(* IEC 61131-3 sources: Mizera_Tube/Plc (part 18) *)

LD   GSTMAC.yChSelMask.3
AND  SEL_ASSE.yExtMask.7
OR(
LD   RemContrCMinus
AND  Rem_Combination
)
OR(
LD   RemContrCPlus
AND  Rem_Combination
)
ST   GESTAX33.xSelected

***************************************
* Change REF quota for ABS reference
***************************************
CAL  RTRIG_AX_SEL33(CLK:=GESTAX33.xSelected)
LD   RTRIG_AX_SEL33.Q
JMPCN NoSel33
LD   ActualQtaAbsRef               ** Absolute homing quota
ST   QtaRefAbsSet                  ** Absolute homing quota setting
NoSel33:

LD   GESTAX33.xSelected
AND  %nvel14.0                     * Se Vale 1 ?gestito "Encoder Assoluto" (Da Configura Asse)
AND (
LD   ActualQtaAbsRef               ** Absolute homing quota
NE   QtaRefAbsSet                  ** Absolute homing quota setting
)
JMPCN NoEq33

LD   QtaRefAbsSet                  ** Absolute homing quota setting
ST   ActualQtaAbsRef               ** Absolute homing quota
NoEq33:
***************************************

LD   Pul_Jogp                      ** (gPlc0.4)jog+ pushbutton
OR(
LD   RemContrCPlus
AND  Rem_Combination
)
AND  EnabJogRTCP                   ** Abilita Jog RTCP
ANDN EMER_GEN                      ** M0.10 Emergenza generale
AND  GESTAX33.xSelected
AND  GESTAX33.xCloseLoop
ST   GESTAX33.xJogPlus

LD   Pul_Jogm                      ** (gPlc0.5)jog- pushbutton
OR(
LD   RemContrCMinus
AND  Rem_Combination
)
AND  EnabJogRTCP                   ** Abilita Jog RTCP
ANDN EMER_GEN                      ** M0.10 Emergenza generale
AND  GESTAX33.xSelected
AND  GESTAX33.xCloseLoop
ST   GESTAX33.xJogMinus

LD   %nvel14.0                     * Se Vale 1 ?gestito "Encoder Assoluto" (Da Configura Asse)
ST   GESTAX33.xZeroForced          * Forzamento asse tarato

LD   AxesHeadNoZeroed              ** Assi Testa non riferiti
OR   BlcAvX1_user                  ** M74.0 Blocco avanzamento asse X1 da user.plc
OR   BlcAvY1_user                  ** M74.4 Blocco avanzamento asse Y da user.plc
OR   CMD_HOLDMOVING_CH3.7          ** M202 Hold moving command axis CH3 (bit0=X, bit1=Y...)
OR   (
LD   %PLCmsg8.9
OR   %PLCerr20.21
ANDN GESTAX33.xJogMinus
)
OR   (
LD   %PLCmsg8.10
ANDN GESTAX33.xJogPlus
)
ST   GESTAX33.xHoldMoving          * Richiesta blocco avanzamento

LD   Res_Axes                      ** (gPlc25.1) reset axes disable electric shaft
ST   GESTAX33.xUnlock

LDN  ch3_in_ref                    ** channel 3 in ref
ANDN EnJogRtcp                     ** (gPlc0.18)Abilitazione Jog RTCP tuning
ST   GESTAX33.xEnFIR               * Abilita filtri FIR
ST   GESTAX33.xEnFrComp            ** Abilita friction compensation

LD   ALWAYS_ZERO                   ** PLCFLAGS.0  Flag sempre stato off
ST   GESTAX33.xDisLimiter

LD   %cn0.rc8.3            * ch0 in alarm
OR   %cn3.rc8.3            * ch3 in alarm
OR   EmerINC
ST   GESTAX33.xSetAlarm     ** Forzamento allarme asse

CAL  GESTAX33

LD   JOGrunning                    ** One axis moving in JOG
OR   %ra19.1         * Stato JOG all'interno del canale
ST   JOGrunning                    ** One axis moving in JOG

LD   REFrunning                    ** One axis moving in REF
OR   %ra19.2
ST   REFrunning                    ** One axis moving in REF

LD   INCrunning                    ** One axis moving in INC
OR   %ra19.3
ST   INCrunning                    ** One axis moving in INC

LD   GESTAX33.yDriveNotEn
S    %PLCerr2.8          * Axis 33, drive not enable

LD   %pa9                * Velocit?massima asse
MUL  1000
DIV  60
ST   %ra50               * Limitazione velocita' massima interpolazione

LD   BSG_INC                       ** rg1.2 Selezione modo INC (inc.fissi)
JMPCN SVIX33

LD   %pa59               * Velocit?di Repos
MUL  1000
DIV  60
MUL  AxesOverride                  ** (gPlc16) feed degli assi (%)
DIV  100
ST   %ra50               * Limitazione velocita' massima interpolazione

SVIX33:
NOAX33:

*******************************************************************************
*   C spindle axis (34)
*******************************************************************************
PATH %ax34
PATH %ax_lsref34

***************************************
*   POWER ON (PON)
***************************************
LD   %pa3.31            * Simulato
ORN  %cn3.cc1.8         * Maschera assi associata al canale
OR(
LD   %nvel11            ** 1=Mechatrolink
EQ   1
AND  %ring.drv1.RDD_wStatus.4 * PON
)
OR(
LD   %nvel11            ** 3,4=CANopen, Ecat
EQ   3
)
OR(
LD   %nvel11            ** 3,4=CANopen, Ecat
EQ   4
)
OR  (
LD   I_I_READY_DRIVE_C             ** Ready signal drive C
AND  (
LD   %ax34.nvel11
EQ   0
)
)
ST   Pon_C                         ** PON Axe C

LD  %cn3.cc1.8           * Maschera assi associata al canale 0
JMPCN NOAX34

***
*   LIMIT SWITCH & REFERENCE SWITCH

LD   %lsrefmode
ST   AXLSREF34.x_REF_mode        * 0=use ref switch...

LD   %lsreflevel
ST   AXLSREF34.x_TYPE_LS         * (1=NC, 0=NO)

LD   I_I_FC_C_NEG                  ** C minimumm limit switch
ST   AXLSREF34.x_MIN_LS          * Min Limit switch

LD   I_I_FC_C_POS                  ** C maximun limit switch
ST   AXLSREF34.x_MAX_LS          * Max Limit switch

LD   I_I_INDEX_C                   ** C1 Axis Homing Switch
ST   AXLSREF34.x_REF_S           * Reference switch

CAL  AXLSREF34

LD   AXLSREF34.y_MIN_LS          * Min Limit switch
ST   GESTAX34.xMinusLS           * Negative limit switch

LD   AXLSREF34.y_MAX_LS          * Max Limit switch
ST   GESTAX34.xPlusLS            * Positive limit switch

LD   AXLSREF34.y_REF_S           * Reference switch
ST   GESTAX34.xRefLS             * Reference
***

LD   TON_ABIL.Q          * Abilitazione drives
ANDN TOF_MALARM.Q        * Assi in allarme
AND  Pon                           ** PON
ANDN CMD_C_C1_OPENLOOP.0             ** M204 Open loop (bit0=1 C, bit1=1 C1)
ST   GESTAX34.xCloseLoop

LD   GSTMAC.yChSelMask.3
AND  SEL_ASSE.yExtMask.8
ST   GESTAX34.xSelected

***************************************
* Change REF quota for ABS reference
***************************************
CAL  RTRIG_AX_SEL34(CLK:=GESTAX34.xSelected)
LD   RTRIG_AX_SEL34.Q
JMPCN NoSel34
LD   ActualQtaAbsRef               ** Absolute homing quota
ST   QtaRefAbsSet                  ** Absolute homing quota setting
NoSel34:

LD   GESTAX34.xSelected
AND  %nvel14.0                     * Se Vale 1 ?gestito "Encoder Assoluto" (Da Configura Asse)
AND (
LD   ActualQtaAbsRef               ** Absolute homing quota
NE   QtaRefAbsSet                  ** Absolute homing quota setting
)
JMPCN NoEq34

LD   QtaRefAbsSet                  ** Absolute homing quota setting
ST   ActualQtaAbsRef               ** Absolute homing quota
NoEq34:
***************************************

LD   JOY_C_P					   **(gPlc2.9)Joystik C + selezionato
OR   (
LD   Pul_Jogp                      ** (gPlc0.4)jog+ pushbutton
AND  GESTAX34.xSelected
)
AND  EnabJogRTCP                   ** Abilita Jog RTCP
ANDN EMER_GEN                      ** M0.10 Emergenza generale
ANDN cmd_c_c1_gear_run
AND  GESTAX34.xCloseLoop
ST   GESTAX34.xJogPlus

LD   JOY_C_M                       **(gPlc2.10)Joystik C - selezionato
OR   (
LD   Pul_Jogm                      ** (gPlc0.5)jog- pushbutton
AND  GESTAX34.xSelected
)
AND  EnabJogRTCP                   ** Abilita Jog RTCP
ANDN EMER_GEN                      ** M0.10 Emergenza generale
ANDN cmd_c_c1_gear_run
AND  GESTAX34.xCloseLoop
ST   GESTAX34.xJogMinus

LD   %nvel14.0                     * Se Vale 1 ?gestito "Encoder Assoluto" (Da Configura Asse)
ST   GESTAX34.xZeroForced          * Forzamento asse tarato

LD   GESTAX5.xHoldMoving           * Richiesta blocco avanzamento
OR   BlcAvX1_user                  ** M74.0 Blocco avanzamento asse X1 da user.plc
OR   HoldSafePipeX                 ** (LsPlc26.2) Hold moving for X axis, not allow manual movement in pipe area
OR   AxesHeadNoZeroed              ** Assi Testa non riferiti
OR   CMD_HOLDMOVING_CH3.8          ** M202 Hold moving command axis CH3 (bit0=X, bit1=Y...)
OR   MOVE_AXIS34.yHoldMov
ST   GESTAX34.xHoldMoving          * Richiesta blocco avanzamento

LD   MOVE_AXIS34.yFromPlc
ST   GESTAX34.xFromPlc

LD   Res_Axes                      ** (gPlc25.1) reset axes disable electric shaft
ST   GESTAX34.xUnlock
ST   O_O_RESET_DRIVE_C             ** C axis drive reset (disable electric shaft)

LDN  ch3_in_ref                    ** channel 3 in ref
ANDN EnJogRtcp                     ** (gPlc0.18)Abilitazione Jog RTCP tuning
ST   GESTAX34.xEnFIR               * Abilita filtri FIR
ST   GESTAX34.xEnFrComp            ** Abilita friction compensation

LD   ALWAYS_ONE
ST   GESTAX34.xDisLimiter

LD   %cn0.rc8.3            * ch0 in alarm
OR   %cn3.rc8.3            * ch3 in alarm
OR   EmerINC
ST   GESTAX34.xSetAlarm     ** Forzamento allarme asse

CAL  GESTAX34

LD   GESTAX34.yDriveNotEn
S    %PLCerr2.4                    * Axis 34, drive not enable

LD   %pa9                * Velocit?massima asse
MUL  1000
DIV  60
ST   %ra50               * Limitazione velocita' massima interpolazione

LD   BSG_INC                       ** rg1.2 Selezione modo INC (inc.fissi)
JMPCN SVIX34

LD   %pa59               * Velocit?di Repos
MUL  1000
DIV  60
MUL  AxesOverride                  ** (gPlc16) feed degli assi (%)
DIV  100
ST   %ra50               * Limitazione velocita' massima interpolazione

SVIX34:
NOAX34:
********************************************************************************

**************************
* Acknowledg funzioni "M"
**************************

LD   R_TRIG10000.Q       ** (M0.8)M10000_CN0: Invoca Unit_1 (inizialavorazione)
OR   R_TRIG10001.Q       ** (M0.9)M10001_CN0: Invoca Unit_1 (finelavorazione)
AND  M30000_CN3                    ** M0.5 M30000_CN3: Attendi Servizio per Unit_1[(M10000 iniziolav.) / M10001(finelav.)]
ORN  Z_Z1_SEL                      ** (gPlc13.6)Testa Z + Z1 selezionata
OR(
LDN  PRGRUN_CN0                    ** M0.0 cn0.rc8.0  Programma in corso
ANDN PRGRUN_CN3                    ** M0.2 cn3.rc8.0  Programma in corso
)
R    BlckM30000_CN3                ** Blocco M30000_CN3 con Z_Z1 selezionati

CAL R_TRIG_M30000CN3(CLK=M30000_CN3) ** Fronte Up M30000CN3

LD   R_TRIG_M30000CN3.Q  ** Fronte Up M30000CN3
OR   F_TRIG10000.Q        ** FronteDwn M10000_CN0: Invoca Unit_1 (inizialavorazione)
OR   F_TRIG10001.Q        ** FronteDwn M10001_CN0: Invoca Unit_1 (finelavorazione)
AND  Z_Z1_SEL                      ** (gPlc13.6)Testa Z + Z1 selezionata
S    BlckM30000_CN3                ** Blocco M30000_CN3 con Z_Z1 selezionati

LD   M30000_CN3                    ** M0.5 M30000_CN3: Attendi Servizio per Unit_1[(M10000 iniziolav.) / M10001(finelav.)]
ANDN Z_Z1_SEL                      ** (gPlc13.6)Testa Z + Z1 selezionata
AND(
LDN  M10000_CN0                    ** M0.8 M10000_CN0: Invoca Unit_1 (inizialavorazione)
ANDN M10001_CN0                    ** M0.9 M10001_CN0: Invoca Unit_1 (finelavorazione)
ORN  HEADZSEL                      ** (gPlc13.4)Testa 1 selezionata
)
ANDN CN3_REQ_VYZ_ISO
OR(
LD   M30000_CN3                    ** M0.5 M30000_CN3: Attendi Servizio per Unit_1[(M10000 iniziolav.) / M10001(finelav.)]
AND  Z_Z1_SEL                      ** (gPlc13.6)Testa Z + Z1 selezionata
AND  BlckM30000_CN3                ** Blocco M30000_CN3 con Z_Z1 selezionati
)
OR(
LD   M30010_CN3                    ** M0.6 Sblocco Richiesta servizio (M10000_CN0 inizialavorazione)
AND  Z_Z1_SEL                      ** (gPlc13.6)Testa Z + Z1 selezionata
ANDN M30010_CN3_4                  ** Blocco M30010_CN3_CN4 con Z_Z1 selezionati
)
OR(
LD   M30011_CN3                    ** M0.7 Sblocco Richiesta servizio (M10001_CN0 finelavorazione)
AND  Z_Z1_SEL                      ** (gPlc13.6)Testa Z + Z1 selezionata
ANDN M30011_CN3_4                  ** Blocco M30011_CN3_CN4 con Z_Z1 selezionati
)
OR   GESTCH3.yWaitMFun
OR   Ack_Mfun_UsrM                 ** (gPlc13.13) Unlock M-Functions from User_M
ST   CH3END.xWaitMFun

CAL  CH3END

*******************************************************************************
*******************************************************************************
*   @@@ CH5: GESTIONE CAMBIO PALLET
*******************************************************************************
*******************************************************************************
PATH %cn5

LD   ALWAYS_ONE                    ** PLCFLAGS.1  Flag sempre stato on
ST   GESTCH5.xCmdFromInput

LD   ALWAYS_ONE                    ** PLCFLAGS.1  Flag sempre stato on
ST   GESTCH5.xEscOpCmd

LD   %PLCFLAGS.0
ST   GESTCH5.xSelFromInput        * Disabilita selezioni standard macchina

LD   Op_Mode0.ySelRef
ST   GESTCH5.xSelREF

LD   Op_Mode0.ySelSingRef
ST   GESTCH0.xSingleRef

LD   Op_Mode0.ySelJog
ST   GESTCH5.xSelJOG

LD   Op_Mode0.ySelInc
ST   GESTCH5.xSelINC

LD   Op_Mode0.ySelMdi
* todo
*AND (
*LD   UP_SELCHAN                    ** ui17 Canale selezionato da monitor canale
*EQ   5
*)
ST   GESTCH5.xSelMDI

LD   Op_Mode0.ySelAut
ST   GESTCH5.xSelAUT

LD   Pul_Start                     ** (gPlc0.1)Start pushbutton
ANDN EMER_GEN                      ** M0.10 Emergenza generale
AND (
LD   BCO_PRGRUN                    ** rc8.0  Programma in corso
AND  BCO_PRGINT                    ** rc8.1  Programma interrotto
AND  ch5_in_aut
OR   ch5_in_ref
OR(
 LD   BCI_MDI                       ** rc0.11  Selettore modi operativi su MDI (semiautom)
 AND (
 LD  UP_SELCHAN                                     ** ui17 Canale selezionato da monitor canale
 EQ  5
 )
)
)
ST   GESTCH5.xStart               * comando START al canale (esterno)

LD   Res_Ch0                       ** (gPlc25.3) reset channel 0
ST   GESTCH5.xReset               * comando RESET al canale (esterno)

LD   %PLCFLAGS.0                  ** Condizioni richiesta hold canale 0
OR(
LD   Pul_Stop                      ** (gPlc0.2)Stop pushbutton
AND  BCI_MDI                       ** rc0.11  Selettore modi operativi su MDI (semiautom)
)
ST   GESTCH5.xHold                * comando Hold al canale (esterno)

LD   GESTCH0.xEmer
ST   GESTCH5.xEmer                * comando Emergenza al canale (esterno)

LD   5555
ST   GESTCH5.xPPNumber            * numero part program da eseguire

LD   %PLCFLAGS.0
ST   GESTCH5.xBlkSearch
ST   GESTCH5.xIntBlkSrc           * Forzam. esec. ricerca blocco interna
ST   GESTCH5.xOverstore  * Ab. overstore dopo ricerca blocco (provv.)

LD   ChannelFeedrate               ** feedrate for channel
ST   GESTCH5.xOverride

CAL  GESTCH5

LD   GESTCH5.yProgramRun          * Programma in corso
ST   PRGRUN_CN5                    ** M0.27 cn5.rc8.0  Programma in corso

LD   BCO_STB_GET                   ** rc8.17 Strobe per GET resources
AND  AxStopSincGRP                 ** (gPlc13.11)Assi Fermi per sincronismo GRP[ax]
ST   BCI_ACK_GET                   ** rc0.29  ACK per GET resource

*******************************************************************************
*   Virtual X axis for tube following algorithm
*******************************************************************************
PATH %ax50
PATH %ax_lsref50

LD  %cc1.0           * Maschera assi associata al canale 0
JMPCN NOAX50

LD   ALWAYS_ZERO                        ** PLCFLAGS.0  Flag sempre stato off
ST   GESTAX50.xMinusLS           * Negative limit switch

LD   ALWAYS_ZERO                      ** PLCFLAGS.0  Flag sempre stato off
ST   GESTAX50.xPlusLS            * Positive limit switch

LD   ALWAYS_ZERO                     ** PLCFLAGS.0  Flag sempre stato off
ST   GESTAX50.xRefLS             * Reference
***

LD   TON_ABIL.Q          * Abilitazione drives
ANDN TOF_MALARM.Q        * Assi in allarme
AND  Pon                           ** PON
ST   GESTAX50.xCloseLoop
ST   GESTAX50_xCloseLoop

LD   ALWAYS_ZERO                   ** PLCFLAGS.0  Flag sempre stato off
ST   GESTAX50.xSelected

LD   ALWAYS_ZERO                   ** PLCFLAGS.0  Flag sempre stato off
ST   GESTAX50.xJogPlus

LD   ALWAYS_ZERO                   ** PLCFLAGS.0  Flag sempre stato off
ST   GESTAX50.xJogMinus

LD   CMD_HOLDMOVING_CH5.0          ** M203 Hold moving command axis CH5 (bit0=X, bit1=Y...)
ST   GESTAX50.xHoldMoving          * Richiesta blocco avanzamento

LD   ALWAYS_ONE                    ** PLCFLAGS.1  Flag sempre stato on
ST   GESTAX50.xZeroForced          * Forzamento asse tarato
ST   GESTAX50.xLockRef    * Blocco avvio ciclo REF da canale

LD   Res_Axes                      ** (gPlc25.1) reset axes disable electric shaft
ST   GESTAX50.xUnlock

LDN  ch5_in_ref                    ** channel 5 in ref
ANDN EnJogRtcp                     ** (gPlc0.18)Abilitazione Jog RTCP tuning
ST   GESTAX50.xEnFIR               * Abilita filtri FIR
ST   GESTAX50.xEnFrComp            ** Abilita friction compensation

LD   ALWAYS_ONE                   ** PLCFLAGS.0  Flag sempre stato off
ST   GESTAX50.xDisLimiter

LD   %cn0.rc8.3            * ch0 in alarm
OR   %cn3.rc8.3            * ch3 in alarm
OR   EmerINC
ST   GESTAX50.xSetAlarm     ** Forzamento allarme asse

CAL  GESTAX50

LD   JOGrunning                    ** One axis moving in JOG
OR   %ra19.1         * Stato JOG all'interno del canale
ST   JOGrunning                    ** One axis moving in JOG

LD   REFrunning                    ** One axis moving in REF
OR   %ra19.2
ST   REFrunning                    ** One axis moving in REF

LD   INCrunning                    ** One axis moving in INC
OR   %ra19.3
ST   INCrunning                    ** One axis moving in INC

LD   %pa9                * Velocit?massima asse
MUL  1000
DIV  60
ST   %ra50               * Limitazione velocita' massima interpolazione

LD   BSG_INC                       ** rg1.2 Selezione modo INC (inc.fissi)
JMPCN SVIX50

LD   %pa59               * Velocit?di Repos
MUL  1000
DIV  60
MUL  AxesOverride                  ** (gPlc16) feed degli assi (%)
DIV  100
ST   %ra50               * Limitazione velocita' massima interpolazione

SVIX50:
NOAX50:

*******************************************************************************
*   Support 1 follower
*******************************************************************************
PATH %ax51
PATH %ax_lsref51

***************************************
*   POWER ON (PON)
***************************************
LD   %pa3.31            * Simulato
ORN  %cc1.1             * Maschera assi associata al canale
OR(
LD   %nvel11            ** 1=Mechatrolink
EQ   1
AND  %ring.drv1.RDD_wStatus.4 * PON
)
OR(
LD   %nvel11            ** 3,4=CANopen, Ecat
EQ   3
)
OR(
LD   %nvel11            ** 3,4=CANopen, Ecat
EQ   4
)
ST   Pon_Z_Follow            ** PON Axe X_T1

LD  %cc1.1           * Maschera assi associata al canale 0
JMPCN NOAX51

***
*   LIMIT SWITCH & REFERENCE SWITCH

LD   %lsrefmode
ST   AXLSREF51.x_REF_mode        * 0=use ref switch...

LD   %lsreflevel
ST   AXLSREF51.x_TYPE_LS         * (1=NC, 0=NO)

LD   I_I_FC_Z1_SUP_NEG
ST   AXLSREF51.x_MIN_LS          * Min Limit switch

LD   I_I_FC_Z1_SUP_POS           * C saw minimumm limit switch
ST   AXLSREF51.x_MAX_LS          * Max Limit switch

LD   ALWAYS_ZERO                   ** PLCFLAGS.0  Flag sempre stato off
ST   AXLSREF51.x_REF_S           * Reference switch

CAL  AXLSREF51

LD   AXLSREF51.y_MIN_LS          * Min Limit switch
ST   GESTAX51.xMinusLS           * Negative limit switch

LD   AXLSREF51.y_MAX_LS          * Max Limit switch
ST   GESTAX51.xPlusLS            * Positive limit switch

LD   AXLSREF51.y_REF_S           * Reference switch
ST   GESTAX51.xRefLS             * Reference
***

LD   TON_ABIL.Q          * Abilitazione drives
ANDN TOF_MALARM.Q        * Assi in allarme
AND  Pon                           ** PON
ST   GESTAX51.xCloseLoop

LD   GSTMAC.yChSelMask.5
AND  SEL_ASSE.yExtMask.1
ST   GESTAX51.xSelected

***************************************
* Change REF quota for ABS reference
***************************************
CAL  RTRIG_AX_SEL51(CLK:=GESTAX51.xSelected)
LD   RTRIG_AX_SEL51.Q
JMPCN NoSel51
LD   ActualQtaAbsRef               ** Absolute homing quota
ST   QtaRefAbsSet                  ** Absolute homing quota setting
NoSel51:

LD   GESTAX51.xSelected
AND  %nvel14.0                     * Se Vale 1 ?gestito "Encoder Assoluto" (Da Configura Asse)
AND (
LD   ActualQtaAbsRef               ** Absolute homing quota
NE   QtaRefAbsSet                  ** Absolute homing quota setting
)
JMPCN NoEq51

LD   QtaRefAbsSet                  ** Absolute homing quota setting
ST   ActualQtaAbsRef               ** Absolute homing quota
NoEq51:

LD   Pul_Jogp                      ** (gPlc0.4)jog+ pushbutton
AND  GESTAX51.xSelected
AND  EnabJogRTCP                   ** Abilita Jog RTCP
ANDN EMER_GEN                      ** M0.10 Emergenza generale
AND  GESTAX51.xCloseLoop
ST   GESTAX51.xJogPlus

LD   Pul_Jogm                      ** (gPlc0.5)jog- pushbutton
AND  GESTAX51.xSelected
AND  EnabJogRTCP                   ** Abilita Jog RTCP
ANDN EMER_GEN                      ** M0.10 Emergenza generale
AND  GESTAX51.xCloseLoop
ST   GESTAX51.xJogMinus

LDN  %ra3.2
OR   %ra0.9
AND  %ra3.13
ST   Supp_51_GoUp

LD   CMD_HOLDMOVING_CH5.1            ** M203 Hold moving command axis CH5 (bit0=X, bit1=Y...)
ST   GESTAX51.xHoldMoving          * Richiesta blocco avanzamento

LD   %nvel14.0                     * Se Vale 1 ?gestito "Encoder Assoluto" (Da Configura Asse)
ST   GESTAX51.xZeroForced          * Forzamento asse tarato

LD   Res_Axes                      ** (gPlc25.1) reset axes disable electric shaft
ST   GESTAX51.xUnlock

LDN  ch5_in_ref                    ** channel 5 in ref
ANDN EnJogRtcp                     ** (gPlc0.18)Abilitazione Jog RTCP tuning
ST   GESTAX51.xEnFIR               * Abilita filtri FIR
ST   GESTAX51.xEnFrComp            ** Abilita friction compensation

LD   ALWAYS_ONE
ST   GESTAX51.xDisLimiter

LD   %cn0.rc8.3                    * ch0 in alarm
OR   %cn3.rc8.3                    * ch3 in alarm
OR   EmerINC
ST   GESTAX51.xSetAlarm            ** Forzamento allarme asse

LD   GRANT5.1
ST   GESTAX51.xFromPlc

CAL  GESTAX51

LD   JOGrunning                    ** One axis moving in JOG
OR   %ra19.1                       * Stato JOG all'interno del canale
ST   JOGrunning                    ** One axis moving in JOG

LD   REFrunning                    ** One axis moving in REF
OR   %ra19.2
ST   REFrunning                    ** One axis moving in REF

LD   INCrunning                    ** One axis moving in INC
OR   %ra19.3
ST   INCrunning                    ** One axis moving in INC

LD   GESTAX51.yDriveNotEn
S    %PLCerr2.15                   * Axis 52, drive not enable

LD   %pa9                          * Velocit?massima asse
MUL  1000
DIV  60
ST   %ra50                         * Limitazione velocita' massima interpolazione

LD   BSG_INC                       ** rg1.2 Selezione modo INC (inc.fissi)
JMPCN SVIX51

LD   %pa59                         * Velocit?di Repos
MUL  1000
DIV  60
MUL  AxesOverride                  ** (gPlc16) feed degli assi (%)
DIV  100
ST   %ra50                         * Limitazione velocita' massima interpolazione

SVIX51:
NOAX51:

* Z 1 real axis for the pipe following algorithm

PATH %ax52
PATH %ax_lsref52

***************************************
*   POWER ON (PON)
***************************************
LD   %pa3.31            * Simulato
ORN  %cc1.2             * Maschera assi associata al canale
OR(
LD   %nvel11            ** 1=Mechatrolink
EQ   1
AND  %ring.drv1.RDD_wStatus.4 * PON
)
OR(
LD   %nvel11            ** 3,4=CANopen, Ecat
EQ   3
)
OR(
LD   %nvel11            ** 3,4=CANopen, Ecat
EQ   4
)
ST   Pon_Z_Follow2            ** PON Axe X_T1

LD  %cc1.2           * Maschera assi associata al canale 0
JMPCN NOAX52

***
*   LIMIT SWITCH & REFERENCE SWITCH

LD   %lsrefmode
ST   AXLSREF52.x_REF_mode        * 0=use ref switch...

LD   %lsreflevel
ST   AXLSREF52.x_TYPE_LS         * (1=NC, 0=NO)

LD   I_I_FC_Z2_SUP_NEG
ST   AXLSREF52.x_MIN_LS          * Min Limit switch

LD   I_I_FC_Z2_SUP_POS           * C saw maximun limit switch
ST   AXLSREF52.x_MAX_LS          * Max Limit switch

LD   ALWAYS_ZERO                   ** PLCFLAGS.0  Flag sempre stato off
ST   AXLSREF52.x_REF_S           * Reference switch

CAL  AXLSREF52

LD   AXLSREF52.y_MIN_LS          * Min Limit switch
ST   GESTAX52.xMinusLS           * Negative limit switch

LD   AXLSREF52.y_MAX_LS          * Max Limit switch
ST   GESTAX52.xPlusLS            * Positive limit switch

LD   AXLSREF52.y_REF_S           * Reference switch
ST   GESTAX52.xRefLS             * Reference
***

LD   TON_ABIL.Q          * Abilitazione drives
ANDN TOF_MALARM.Q        * Assi in allarme
AND  Pon                           ** PON
ST   GESTAX52.xCloseLoop

LD   GSTMAC.yChSelMask.5
AND  SEL_ASSE.yExtMask.2
ST   GESTAX52.xSelected

***************************************
* Change REF quota for ABS reference
***************************************
CAL  RTRIG_AX_SEL52(CLK:=GESTAX52.xSelected)
LD   RTRIG_AX_SEL52.Q
JMPCN NoSel52
LD   ActualQtaAbsRef               ** Absolute homing quota
ST   QtaRefAbsSet                  ** Absolute homing quota setting
NoSel52:

LD   GESTAX52.xSelected
AND  %nvel14.0                     * Se Vale 1 ?gestito "Encoder Assoluto" (Da Configura Asse)
AND (
LD   ActualQtaAbsRef               ** Absolute homing quota
NE   QtaRefAbsSet                  ** Absolute homing quota setting
)
JMPCN NoEq52

LD   QtaRefAbsSet                  ** Absolute homing quota setting
ST   ActualQtaAbsRef               ** Absolute homing quota
NoEq52:
***************************************

LD   Pul_Jogp                      ** (gPlc0.4)jog+ pushbutton
AND  GESTAX52.xSelected
AND  EnabJogRTCP                   ** Abilita Jog RTCP
ANDN EMER_GEN                      ** M0.10 Emergenza generale
AND  GESTAX52.xCloseLoop
ST   GESTAX52.xJogPlus

LD   Pul_Jogm                      ** (gPlc0.5)jog- pushbutton
AND  GESTAX52.xSelected
AND  EnabJogRTCP                   ** Abilita Jog RTCP
ANDN EMER_GEN                      ** M0.10 Emergenza generale
AND  GESTAX52.xCloseLoop
ST   GESTAX52.xJogMinus

LDN  %ra3.2
OR   %ra0.9
AND  %ra3.13
ST   Supp_52_GoUp

LD   CMD_HOLDMOVING_CH5.2            ** M203 Hold moving command axis CH5 (bit0=X, bit1=Y...)
ST   GESTAX52.xHoldMoving          * Richiesta blocco avanzamento

LD   %nvel14.0                     * Se Vale 1 ?gestito "Encoder Assoluto" (Da Configura Asse)
ST   GESTAX52.xZeroForced          * Forzamento asse tarato

LD   Res_Axes                      ** (gPlc25.1) reset axes disable electric shaft
ST   GESTAX52.xUnlock

LDN  ch5_in_ref                    ** channel 5 in ref
ANDN EnJogRtcp                     ** (gPlc0.18)Abilitazione Jog RTCP tuning
ST   GESTAX52.xEnFIR               * Abilita filtri FIR
ST   GESTAX52.xEnFrComp            ** Abilita friction compensation

LD   ALWAYS_ONE
ST   GESTAX52.xDisLimiter

LD   %cn0.rc8.3            * ch0 in alarm
OR   %cn3.rc8.3            * ch3 in alarm
OR   EmerINC
ST   GESTAX52.xSetAlarm     ** Forzamento allarme asse

LD   GRANT5.2
ST   GESTAX52.xFromPlc

CAL  GESTAX52

LD   JOGrunning                    ** One axis moving in JOG
OR   %ra19.1         * Stato JOG all'interno del canale
ST   JOGrunning                    ** One axis moving in JOG

LD   REFrunning                    ** One axis moving in REF
OR   %ra19.2
ST   REFrunning                    ** One axis moving in REF

LD   INCrunning                    ** One axis moving in INC
OR   %ra19.3
ST   INCrunning                    ** One axis moving in INC

LD   GESTAX52.yDriveNotEn
S    %PLCerr2.14                    * Axis 52, drive not enable

LD   %pa9                * Velocit?massima asse
MUL  1000
DIV  60
ST   %ra50               * Limitazione velocita' massima interpolazione

LD   BSG_INC                       ** rg1.2 Selezione modo INC (inc.fissi)
JMPCN SVIX52

LD   %pa59               * Velocit?di Repos
MUL  1000
DIV  60
MUL  AxesOverride                  ** (gPlc16) feed degli assi (%)
DIV  100
ST   %ra50               * Limitazione velocita' massima interpolazione

SVIX52:
NOAX52:

* Z 3 real axis for the pipe following algorithm

PATH %ax53
PATH %ax_lsref53

***************************************
*   POWER ON (PON)
***************************************
LD   %pa3.31            * Simulato
ORN  %cc1.2             * Maschera assi associata al canale
OR(
LD   %nvel11            ** 1=Mechatrolink
EQ   1
AND  %ring.drv1.RDD_wStatus.4 * PON
)
OR(
LD   %nvel11            ** 3,4=CANopen, Ecat
EQ   3
)
OR(
LD   %nvel11            ** 3,4=CANopen, Ecat
EQ   4
)
OR  (
LD   I_I_READY_DRIVE_Z_FOLL        ** Ready signal drive Z_follower
AND  (
LD   %ax52.nvel11
EQ   0
)
)
ST   Pon_Z_Follow3           ** PON Axe X_T1

LD  %cc1.3           * Maschera assi associata al canale 0
JMPCN NOAX53

***
*   LIMIT SWITCH & REFERENCE SWITCH

LD   %lsrefmode
ST   AXLSREF53.x_REF_mode        * 0=use ref switch...

LD   %lsreflevel
ST   AXLSREF53.x_TYPE_LS         * (1=NC, 0=NO)

LD   I_I_FC_Z3_SUP_NEG                   ** PLCFLAGS.0  Flag sempre stato off
ST   AXLSREF53.x_MIN_LS          * Min Limit switch

LD   I_I_FC_Z3_SUP_POS           * C saw maximun limit switch
ST   AXLSREF53.x_MAX_LS          * Max Limit switch

LD   ALWAYS_ZERO                   ** PLCFLAGS.0  Flag sempre stato off
ST   AXLSREF53.x_REF_S           * Reference switch

CAL  AXLSREF53

LD   AXLSREF53.y_MIN_LS          * Min Limit switch
ST   GESTAX53.xMinusLS           * Negative limit switch

LD   AXLSREF53.y_MAX_LS          * Max Limit switch
ST   GESTAX53.xPlusLS            * Positive limit switch

LD   AXLSREF53.y_REF_S           * Reference switch
ST   GESTAX53.xRefLS             * Reference
***

LD   TON_ABIL.Q          * Abilitazione drives
ANDN TOF_MALARM.Q        * Assi in allarme
AND  Pon                           ** PON
ST   GESTAX53.xCloseLoop

LD   GSTMAC.yChSelMask.5
AND  SEL_ASSE.yExtMask.3
ST   GESTAX53.xSelected

***************************************
* Change REF quota for ABS reference
***************************************
CAL  RTRIG_AX_SEL53(CLK:=GESTAX53.xSelected)
LD   RTRIG_AX_SEL53.Q
JMPCN NoSel53
LD   ActualQtaAbsRef               ** Absolute homing quota
ST   QtaRefAbsSet                  ** Absolute homing quota setting
NoSel53:

LD   GESTAX53.xSelected
AND  %nvel14.0                     * Se Vale 1 ?gestito "Encoder Assoluto" (Da Configura Asse)
AND (
LD   ActualQtaAbsRef               ** Absolute homing quota
NE   QtaRefAbsSet                  ** Absolute homing quota setting
)
JMPCN NoEq53

LD   QtaRefAbsSet                  ** Absolute homing quota setting
ST   ActualQtaAbsRef               ** Absolute homing quota
NoEq53:
***************************************

LD   Pul_Jogp                      ** (gPlc0.4)jog+ pushbutton
AND  GESTAX53.xSelected
AND  EnabJogRTCP                   ** Abilita Jog RTCP
ANDN EMER_GEN                      ** M0.10 Emergenza generale
AND  GESTAX53.xCloseLoop
ST   GESTAX53.xJogPlus

LD   Pul_Jogm                      ** (gPlc0.5)jog- pushbutton
AND  GESTAX53.xSelected
AND  EnabJogRTCP                   ** Abilita Jog RTCP
ANDN EMER_GEN                      ** M0.10 Emergenza generale
AND  GESTAX53.xCloseLoop
ST   GESTAX53.xJogMinus

LDN  %ra3.2
OR   %ra0.9
AND  %ra3.13
ST   Supp_53_GoUp

LD   CMD_HOLDMOVING_CH5.3            ** M203 Hold moving command axis CH5 (bit0=X, bit1=Y...)
ST   GESTAX53.xHoldMoving          * Richiesta blocco avanzamento

LD   %nvel14.0                     * Se Vale 1 ?gestito "Encoder Assoluto" (Da Configura Asse)
ST   GESTAX53.xZeroForced          * Forzamento asse tarato

LD   Res_Axes                      ** (gPlc25.1) reset axes disable electric shaft
ST   GESTAX53.xUnlock

LDN  ch5_in_ref                    ** channel 5 in ref
ANDN EnJogRtcp                     ** (gPlc0.18)Abilitazione Jog RTCP tuning
ST   GESTAX53.xEnFIR               * Abilita filtri FIR
ST   GESTAX53.xEnFrComp            ** Abilita friction compensation

LD   ALWAYS_ONE
ST   GESTAX53.xDisLimiter

LD   %cn0.rc8.3            * ch0 in alarm
OR   %cn3.rc8.3            * ch3 in alarm
OR   EmerINC
ST   GESTAX53.xSetAlarm     ** Forzamento allarme asse

LD   GRANT5.3
ST   GESTAX53.xFromPlc

CAL  GESTAX53

LD   JOGrunning                    ** One axis moving in JOG
OR   %ra19.1         * Stato JOG all'interno del canale
ST   JOGrunning                    ** One axis moving in JOG

LD   REFrunning                    ** One axis moving in REF
OR   %ra19.2
ST   REFrunning                    ** One axis moving in REF

LD   INCrunning                    ** One axis moving in INC
OR   %ra19.3
ST   INCrunning                    ** One axis moving in INC

LD   GESTAX53.yDriveNotEn
S    %PLCerr2.17                   * Axis 53, drive not enable

LD   %pa9                * Velocit?massima asse
MUL  1000
DIV  60
ST   %ra50               * Limitazione velocita' massima interpolazione

LD   BSG_INC                       ** rg1.2 Selezione modo INC (inc.fissi)
JMPCN SVIX53

LD   %pa59               * Velocit?di Repos
MUL  1000
DIV  60
MUL  AxesOverride                  ** (gPlc16) feed degli assi (%)
DIV  100
ST   %ra50               * Limitazione velocita' massima interpolazione

SVIX53:
NOAX53:

* Z 4 real axis for the pipe following algorithm

PATH %ax54
PATH %ax_lsref54

***************************************
*   POWER ON (PON)
***************************************
LD   %pa3.31            * Simulato
ORN  %cc1.4             * Maschera assi associata al canale
OR(
LD   %nvel11            ** 1=Mechatrolink
EQ   1
AND  %ring.drv1.RDD_wStatus.4 * PON
)
OR(
LD   %nvel11            ** 3,4=CANopen, Ecat
EQ   3
)
OR(
LD   %nvel11            ** 3,4=CANopen, Ecat
EQ   4
)
ST   Pon_Z_Follow4           ** PON Axe X_T1

LD  %cc1.4           * Maschera assi associata al canale 0
JMPCN NOAX54

***
*   LIMIT SWITCH & REFERENCE SWITCH

LD   %lsrefmode
ST   AXLSREF54.x_REF_mode        * 0=use ref switch...

LD   %lsreflevel
ST   AXLSREF54.x_TYPE_LS         * (1=NC, 0=NO)

LD   I_I_FC_Z4_SUP_NEG                   ** PLCFLAGS.0  Flag sempre stato off
ST   AXLSREF54.x_MIN_LS          * Min Limit switch

LD   I_I_FC_Z4_SUP_POS           * C saw minimumm limit switch
ST   AXLSREF54.x_MAX_LS          * Max Limit switch

LD   ALWAYS_ZERO                   ** PLCFLAGS.0  Flag sempre stato off
ST   AXLSREF54.x_REF_S           * Reference switch

CAL  AXLSREF54

LD   AXLSREF54.y_MIN_LS          * Min Limit switch
ST   GESTAX54.xMinusLS           * Negative limit switch

LD   AXLSREF54.y_MAX_LS          * Max Limit switch
ST   GESTAX54.xPlusLS            * Positive limit switch

LD   AXLSREF54.y_REF_S           * Reference switch
ST   GESTAX54.xRefLS             * Reference
***

LD   TON_ABIL.Q          * Abilitazione drives
ANDN TOF_MALARM.Q        * Assi in allarme
AND  Pon                           ** PON
ST   GESTAX54.xCloseLoop

LD   GSTMAC.yChSelMask.5
AND  SEL_ASSE.yExtMask.4
ST   GESTAX54.xSelected

***************************************
* Change REF quota for ABS reference
***************************************
CAL  RTRIG_AX_SEL54(CLK:=GESTAX54.xSelected)
LD   RTRIG_AX_SEL54.Q
JMPCN NoSel54
LD   ActualQtaAbsRef               ** Absolute homing quota
ST   QtaRefAbsSet                  ** Absolute homing quota setting
NoSel54:

LD   GESTAX54.xSelected
AND  %nvel14.0                     * Se Vale 1 ?gestito "Encoder Assoluto" (Da Configura Asse)
AND (
LD   ActualQtaAbsRef               ** Absolute homing quota
NE   QtaRefAbsSet                  ** Absolute homing quota setting
)
JMPCN NoEq54

LD   QtaRefAbsSet                  ** Absolute homing quota setting
ST   ActualQtaAbsRef               ** Absolute homing quota
NoEq54:
***************************************

LD   Pul_Jogp                      ** (gPlc0.4)jog+ pushbutton
AND  GESTAX54.xSelected
AND  EnabJogRTCP                   ** Abilita Jog RTCP
ANDN EMER_GEN                      ** M0.10 Emergenza generale
AND  GESTAX54.xCloseLoop
ST   GESTAX54.xJogPlus

LD   Pul_Jogm                      ** (gPlc0.5)jog- pushbutton
AND  GESTAX54.xSelected
AND  EnabJogRTCP                   ** Abilita Jog RTCP
ANDN EMER_GEN                      ** M0.10 Emergenza generale
AND  GESTAX54.xCloseLoop
ST   GESTAX54.xJogMinus

LD   CMD_HOLDMOVING_CH5.4            ** M203 Hold moving command axis CH5 (bit0=X, bit1=Y...)
ST   GESTAX54.xHoldMoving          * Richiesta blocco avanzamento

LD   %nvel14.0                     * Se Vale 1 ?gestito "Encoder Assoluto" (Da Configura Asse)
ST   GESTAX54.xZeroForced          * Forzamento asse tarato

LD   Res_Axes                      ** (gPlc25.1) reset axes disable electric shaft
ST   GESTAX54.xUnlock

LDN  ch5_in_ref                    ** channel 5 in ref
ANDN EnJogRtcp                     ** (gPlc0.18)Abilitazione Jog RTCP tuning
ST   GESTAX54.xEnFIR               * Abilita filtri FIR
ST   GESTAX54.xEnFrComp            ** Abilita friction compensation

LD   ALWAYS_ONE
ST   GESTAX54.xDisLimiter

LD   %cn0.rc8.3            * ch0 in alarm
OR   %cn3.rc8.3            * ch3 in alarm
OR   EmerINC
ST   GESTAX54.xSetAlarm     ** Forzamento allarme asse

LD   GRANT5.4
ST   GESTAX54.xFromPlc

CAL  GESTAX54

LD   JOGrunning                    ** One axis moving in JOG
OR   %ra19.1         * Stato JOG all'interno del canale
ST   JOGrunning                    ** One axis moving in JOG

LD   REFrunning                    ** One axis moving in REF
OR   %ra19.2
ST   REFrunning                    ** One axis moving in REF

LD   INCrunning                    ** One axis moving in INC
OR   %ra19.3
ST   INCrunning                    ** One axis moving in INC

LD   GESTAX54.yDriveNotEn
S    %PLCerr2.18                    * Axis 52, drive not enable

LD   %pa9                * Velocit?massima asse
MUL  1000
DIV  60
ST   %ra50               * Limitazione velocita' massima interpolazione

LD   BSG_INC                       ** rg1.2 Selezione modo INC (inc.fissi)
JMPCN SVIX54

LD   %pa59               * Velocit?di Repos
MUL  1000
DIV  60
MUL  AxesOverride                  ** (gPlc16) feed degli assi (%)
DIV  100
ST   %ra50               * Limitazione velocita' massima interpolazione

SVIX54:
NOAX54:

*******************************************************************************
*   Spindles safe gearing reset
*******************************************************************************
CAL  TOF_RESET_GEAR(IN=Pul_Reset, PT=50)
LDN  %cn0.rc8.0
ST   appoggio
CAL  TP_PRGOFF_GEAR(IN=appoggio, PT=50)

*******************************************************************************
*   C1 spindle axis (57)
*******************************************************************************
PATH %ax57
PATH %ax_lsref57

***************************************
*   POWER ON (PON)
***************************************
LD   %pa3.31            * Simulato
ORN  %cc1.7             * Maschera assi associata al canale
OR(
LD   %nvel11            ** 1=Mechatrolink
EQ   1
AND  %ring.drv1.RDD_wStatus.4 * PON
)
OR(
LD   %nvel11            ** 3,4=CANopen, Ecat
EQ   3
)
OR(
LD   %nvel11            ** 3,4=CANopen, Ecat
EQ   4
)
OR   (
LD   I_I_READY_DRIVE_C1            ** Ready signal drive C1
AND  (
LD   %ax54.nvel11
EQ   0
)
)
ST   Pon_C1                        ** PON Axe C1

LD  %cn5.cc1.7           * Maschera assi associata al canale 0
JMPCN NOAX57

***
*   LIMIT SWITCH & REFERENCE SWITCH

LD   %lsrefmode
ST   AXLSREF57.x_REF_mode        * 0=use ref switch...

LD   %lsreflevel
ST   AXLSREF57.x_TYPE_LS         * (1=NC, 0=NO)

LD   I_I_FC_C1_NEG                 ** C1 minimumm limit switch
ST   AXLSREF57.x_MIN_LS          * Min Limit switch

LD   I_I_FC_C1_POS                 ** C1 maximun limit switch
ST   AXLSREF57.x_MAX_LS          * Max Limit switch

LD   I_I_INDEX_C1                  ** C1 Axis Homing Switch
ST   AXLSREF57.x_REF_S           * Reference switch

CAL  AXLSREF57

LD   AXLSREF57.y_MIN_LS          * Min Limit switch
ST   GESTAX57.xMinusLS           * Negative limit switch

LD   AXLSREF57.y_MAX_LS          * Max Limit switch
ST   GESTAX57.xPlusLS            * Positive limit switch

LD   AXLSREF57.y_REF_S           * Reference switch
ST   GESTAX57.xRefLS             * Reference
***

LD   TON_ABIL.Q          * Abilitazione drives
ANDN TOF_MALARM.Q        * Assi in allarme
AND  Pon                           ** PON
ANDN CMD_C_C1_OPENLOOP.1           ** M204 Open loop (bit0=1 C, bit1=1 C1)
ST   GESTAX57.xCloseLoop

LD   GSTMAC.yChSelMask.5
AND  SEL_ASSE.yExtMask.7
ANDN spindle_geared                ** axes gearing enable from function block
ST   GESTAX57.xSelected

***************************************
* Change REF quota for ABS reference
***************************************
CAL  RTRIG_AX_SEL57(CLK:=GESTAX57.xSelected)
LD   RTRIG_AX_SEL57.Q
JMPCN NoSel57
LD   ActualQtaAbsRef               ** Absolute homing quota
ST   QtaRefAbsSet                  ** Absolute homing quota setting
NoSel57:

LD   GESTAX57.xSelected
AND  %nvel14.0                     * Se Vale 1 ?gestito "Encoder Assoluto" (Da Configura Asse)
AND (
LD   ActualQtaAbsRef               ** Absolute homing quota
NE   QtaRefAbsSet                  ** Absolute homing quota setting
)
JMPCN NoEq57

LD   QtaRefAbsSet                  ** Absolute homing quota setting
ST   ActualQtaAbsRef               ** Absolute homing quota
NoEq57:
***************************************

LD   Pul_Jogp                      ** (gPlc0.4)jog+ pushbutton
AND  EnabJogRTCP                   ** Abilita Jog RTCP
ANDN cmd_c_c1_gear_run
AND  GESTAX57.xSelected
ST   GESTAX57.xJogPlus

LD   Pul_Jogm                      ** (gPlc0.5)jog- pushbutton
AND  EnabJogRTCP                   ** Abilita Jog RTCP
ANDN cmd_c_c1_gear_run
AND  GESTAX57.xSelected
ST   GESTAX57.xJogMinus

LD   %nvel14.0                     * Se Vale 1 ?gestito "Encoder Assoluto" (Da Configura Asse)
ST   GESTAX57.xZeroForced          * Forzamento asse tarato

LD   GESTAX5.xHoldMoving           * Richiesta blocco avanzamento
OR   BlcAvX1_user                  ** M74.0 Blocco avanzamento asse X1 da user.plc
OR   AxesHeadNoZeroed              ** Assi Testa non riferiti
OR   CMD_HOLDMOVING_CH5.7          ** M203 Hold moving command axis CH5 (bit0=X, bit1=Y...)
OR(
 LD   GESTAX34.xHoldMoving          * Richiesta blocco avanzamento
 AND  spindle_geared                ** axes gearing enable from function block
)
ST   GESTAX57.xHoldMoving          * Richiesta blocco avanzamento

LD   GEAR_C_C1.xax_ENABLE
OR   start_alignment
AND  GESTAX57.xCloseLoop
ST   GESTAX57.xFromPlc

LD   Res_Axes                      ** (gPlc25.1) reset axes disable electric shaft
ST   GESTAX57.xUnlock
ST   O_O_RESET_DRIVE_C1            ** C1 axis drive reset (disable electric shaft)

LDN  ch5_in_ref                    ** channel 5 in ref
ANDN EnJogRtcp                     ** (gPlc0.18)Abilitazione Jog RTCP tuning
ST   GESTAX57.xEnFIR               * Abilita filtri FIR
ST   GESTAX57.xEnFrComp            ** Abilita friction compensation

LD   ALWAYS_ONE
ST   GESTAX57.xDisLimiter

LD   %cn0.rc8.3            * ch0 in alarm
OR   %cn3.rc8.3            * ch3 in alarm
OR   EmerINC
ST   GESTAX57.xSetAlarm     ** Forzamento allarme asse

CAL  GESTAX57

LD   GESTAX57.yDriveNotEn
S    %PLCerr2.6                    * Axis 54, drive not enable

LD   %pa9                * Velocit?massima asse
MUL  1000
DIV  60
ST   %ra50               * Limitazione velocita' massima interpolazione

LD   BSG_INC                       ** rg1.2 Selezione modo INC (inc.fissi)
JMPCN SVIX57

LD   %pa59               * Velocit?di Repos
MUL  1000
DIV  60
MUL  AxesOverride                  ** (gPlc16) feed degli assi (%)
DIV  100
ST   %ra50               * Limitazione velocita' massima interpolazione

SVIX57:

LD  Pon                            ** PON
AND GESTAX34.xCloseLoop  * condition for real an simulation machine
AND GESTAX57.xCloseLoop  * condition for real an simulation machine
ST  appoggio                       ** Appoggio

CAL RTRIG_PON (CLK:=appoggio)      ** Appoggio

LD  Manual_alignment
AND appoggio
ST  Manual_align

CAL RTRIG_man_ali(CLK:=Manual_align)

LD   RTRIG_PON.Q
AND  (
LD   %ax34.ra4
SUB  %ax57.ra4
ABS
GT   200                 * threshold 1 dmm
AND (
 LD   %ax34.ra4
 SUB  %ax57.ra4
 ABS
 LE   %LSRCostK8
)
)
OR   RTRIG_man_ali.Q
AND  MACC_TARATA                   ** (gPlc0.9)Assi tarati
AND  %ax34.ra3.0                    * Asse fermo teorico
AND  %ax57.ra3.0                    * Asse fermo teorico
ANDN PRGRUN_CN0                    ** M0.0 cn0.rc8.0  Programma in corso
S    start_alignment

LD   start_alignment
ST   POS_AX57.xax_ENABLE

LDN  POS_AX57.xax_ENABLE
OR   TP_PRGOFF_GEAR.Q
OR   TOF_RESET_GEAR.Q
ST   POS_AX57.xax_CLEAR

LD   POS_AX57.xax_ENABLE
AND  POS_AX57.yax_READY
ANDN POS_AX57.yax_ENDOK
ANDN POS_AX57.yax_ENDERR
ST   POS_AX57.xax_START

LD   %ax34.ra4
ST   POS_AX57.xax_QUOTA

LD   %pa9
ST   POS_AX57.xax_VEL

CAL  POS_AX57

LD   POS_AX57.yax_ENDOK
OR   POS_AX57.yax_ENDERR
OR   I_I_EMERGENZA                 ** Machine OK (no EMERG.)
***OR   EMER_GEN                      ** (M0.10)Emergenza generale
R    start_alignment

LD   %ax34.ra4
SUB  %ax57.ra4
ABS
GT   %LSRCostK8
AND  PRGRUN_CN0                    ** M0.0 cn0.rc8.0  Programma in corso
ANDN %ServiceMillePGM.1
S   %PLCerr0.31                    * Spindles not aligned

LD  Pul_Reset                      ** (gPlc0.3)Reset pushbutton
R   %PLCerr0.31                    * Spindles not aligned

NOAX57:

LD  Pul_Reset                      ** (gPlc0.3)Reset pushbutton
R   GearingC_C1Off

***
* Gearing C-C1
LD   CMD_C_C1_UNLOCK
EQ   1
OR   GearingC_C1Off
ST   appoggio

CAL  TRIG_GEAR_C_C1(CLK:=appoggio)

LDN  EMER_GEN                      ** M0.10 Emergenza generale
AND  GESTAX57.xCloseLoop
ANDN POS_AX57.xax_ENABLE
ANDN ch5_in_ref                    ** channel 5 in ref
ST   appoggio

LD   appoggio
ANDN CMD_C_C1_UNLOCK
S    cmd_c_c1_gear_run

LD   spindle_geared                ** axes gearing enable from function block
OR   CMD_C_C1_UNLOCK
R    cmd_c_c1_gear_run

CAL  TON_GEAR_C_C1(IN=appoggio,PT=800) ** Appoggio

LD   TON_GEAR_C_C1.Q
ANDN ch0_in_ref                    ** channel 0 in ref
ANDN BUP_JOGOPEN                   ** ui16.16 Selezione esecuzione JOG a loop aperto
AND (
LDN  CMD_C_C1_UNLOCK               ** M200 Unlock gearing C-C1
ANDN GearingC_C1Off
)
ST   GEAR_C_C1.xax_ENABLE          * ------> CONDIZ.RICHIESTA DI AGGANCIO

LDN  GEAR_C_C1.xax_ENABLE
OR   TRIG_GEAR_C_C1.Q
OR   TP_PRGOFF_GEAR.Q
OR   TOF_RESET_GEAR.Q
ST   GEAR_C_C1.xax_CLEAR

LD   GEAR_C_C1.xax_ENABLE
AND  GEAR_C_C1.yax_READY
ANDN GEAR_C_C1.yax_ENDOK
ANDN GEAR_C_C1.yax_ENDERR
ST   GEAR_C_C1.xax_START

LD   34
ST   GEAR_C_C1.xax_MASTER

LD   1                             * Modalit?di inseguimente(VA BENE LASCIARE SEMPRE 1)
ST   GEAR_C_C1.xax_TRNUM
ST   GEAR_C_C1.xax_TRDEN

CAL  GEAR_C_C1

LD   GEAR_C_C1.yax_RUNNING
AND  GEAR_C_C1.xax_ENABLE
S    spindle_geared                ** axes gearing enable from function block

LDN  GEAR_C_C1.xax_ENABLE
OR   GEAR_C_C1.yax_ENDERR
R    spindle_geared                ** axes gearing enable from function block

LDN  spindle_geared                ** axes gearing enable from function block
ST   FBK_C_C1_UNLOCK               ** M201 Feedback gearing C-C1

*******************************************************************************
*   C2 spindle axis (58)
*******************************************************************************
PATH %ax58
PATH %ax_lsref58

***************************************
*   POWER ON (PON)
***************************************
LD   %pa3.31            * Simulato
ORN  %cc1.8             * Maschera assi associata al canale
OR(
LD   %nvel11            ** 1=Mechatrolink
EQ   1
AND  %ring.drv1.RDD_wStatus.4 * PON
)
OR(
LD   %nvel11            ** 3,4=CANopen, Ecat
EQ   3
)
OR(
LD   %nvel11            ** 3,4=CANopen, Ecat
EQ   4
)
OR   (
LD   I_I_READY_DRIVE_C2            ** Ready signal drive C1
AND  (
LD   %ax58.nvel11
EQ   0
)
)
ST   Pon_C2                        ** PON Axe C1

LD  %cn5.cc1.8           * Maschera assi associata al canale 0
JMPCN NOAX58

***
*   LIMIT SWITCH & REFERENCE SWITCH

LD   %lsrefmode
ST   AXLSREF58.x_REF_mode        * 0=use ref switch...

LD   %lsreflevel
ST   AXLSREF58.x_TYPE_LS         * (1=NC, 0=NO)

LD   I_I_FC_C2_NEG                 ** C1 minimumm limit switch
ST   AXLSREF58.x_MIN_LS          * Min Limit switch

LD   I_I_FC_C2_POS                 ** C1 maximun limit switch
ST   AXLSREF58.x_MAX_LS          * Max Limit switch

LD   I_I_INDEX_C2                  ** C1 Axis Homing Switch
ST   AXLSREF58.x_REF_S           * Reference switch

CAL  AXLSREF58

LD   AXLSREF58.y_MIN_LS          * Min Limit switch
ST   GESTAX58.xMinusLS           * Negative limit switch

LD   AXLSREF58.y_MAX_LS          * Max Limit switch
ST   GESTAX58.xPlusLS            * Positive limit switch

LD   AXLSREF58.y_REF_S           * Reference switch
ST   GESTAX58.xRefLS             * Reference
***

LD   TON_ABIL.Q          * Abilitazione drives
ANDN TOF_MALARM.Q        * Assi in allarme
AND  Pon                           ** PON
ANDN CMD_C_C1_OPENLOOP.2           ** M204 Open loop (bit0=1 C, bit1=1 C1)
ST   GESTAX58.xCloseLoop

LD   GSTMAC.yChSelMask.5
AND  SEL_ASSE.yExtMask.8
ANDN spindle_geared_C2                ** axes gearing enable from function block
ST   GESTAX58.xSelected

***************************************
* Change REF quota for ABS reference
***************************************
CAL  RTRIG_AX_SEL58(CLK:=GESTAX58.xSelected)
LD   RTRIG_AX_SEL58.Q
JMPCN NoSel58
LD   ActualQtaAbsRef               ** Absolute homing quota
ST   QtaRefAbsSet                  ** Absolute homing quota setting
NoSel58:

LD   GESTAX58.xSelected
AND  %nvel14.0                     * Se Vale 1 ?gestito "Encoder Assoluto" (Da Configura Asse)
AND (
LD   ActualQtaAbsRef               ** Absolute homing quota
NE   QtaRefAbsSet                  ** Absolute homing quota setting
)
JMPCN NoEq58

LD   QtaRefAbsSet                  ** Absolute homing quota setting
ST   ActualQtaAbsRef               ** Absolute homing quota
NoEq58:
***************************************

LD   Pul_Jogp                      ** (gPlc0.4)jog+ pushbutton
AND  EnabJogRTCP                   ** Abilita Jog RTCP
ANDN cmd_c_c2_gear_run
AND  GESTAX58.xSelected
ST   GESTAX58.xJogPlus

LD   Pul_Jogm                      ** (gPlc0.5)jog- pushbutton
AND  EnabJogRTCP                   ** Abilita Jog RTCP
ANDN cmd_c_c2_gear_run
AND  GESTAX58.xSelected
ST   GESTAX58.xJogMinus

LD   %nvel14.0                     * Se Vale 1 ?gestito "Encoder Assoluto" (Da Configura Asse)
ST   GESTAX58.xZeroForced          * Forzamento asse tarato

LD   GESTAX5.xHoldMoving           * Richiesta blocco avanzamento
OR   BlcAvX1_user                  ** M74.0 Blocco avanzamento asse X1 da user.plc
OR   AxesHeadNoZeroed              ** Assi Testa non riferiti
OR   CMD_HOLDMOVING_CH5.7          ** M203 Hold moving command axis CH5 (bit0=X, bit1=Y...)
OR(
 LD   GESTAX34.xHoldMoving          * Richiesta blocco avanzamento
 AND  spindle_geared_C2                ** axes gearing enable from function block
)
ST   GESTAX58.xHoldMoving          * Richiesta blocco avanzamento

LD   GEAR_C_C2.xax_ENABLE
OR   start_alignment_C2
AND  GESTAX58.xCloseLoop
ST   GESTAX58.xFromPlc

LD   Res_Axes                      ** (gPlc25.1) reset axes disable electric shaft
ST   GESTAX58.xUnlock
ST   O_O_RESET_DRIVE_C2            ** C2 axis drive reset (disable electric shaft)

LDN  ch5_in_ref                    ** channel 5 in ref
ANDN EnJogRtcp                     ** (gPlc0.18)Abilitazione Jog RTCP tuning
ST   GESTAX58.xEnFIR               * Abilita filtri FIR
ST   GESTAX58.xEnFrComp            ** Abilita friction compensation

LD   ALWAYS_ONE
ST   GESTAX58.xDisLimiter

LD   %cn0.rc8.3            * ch0 in alarm
OR   %cn3.rc8.3            * ch3 in alarm
OR   EmerINC
ST   GESTAX58.xSetAlarm     ** Forzamento allarme asse

CAL  GESTAX58

LD   GESTAX58.yDriveNotEn
S    %PLCerr2.16                    * Axis 55, drive not enable

LD   %pa9                * Velocit?massima asse
MUL  1000
DIV  60
ST   %ra50               * Limitazione velocita' massima interpolazione

LD   BSG_INC                       ** rg1.2 Selezione modo INC (inc.fissi)
JMPCN SVIX58

LD   %pa59               * Velocit?di Repos
MUL  1000
DIV  60
MUL  AxesOverride                  ** (gPlc16) feed degli assi (%)
DIV  100
ST   %ra50               * Limitazione velocita' massima interpolazione

SVIX58:

LD  Pon                            ** PON
AND GESTAX34.xCloseLoop  * condition for real an simulation machine
AND GESTAX58.xCloseLoop  * condition for real an simulation machine
ST  appoggio                       ** Appoggio

CAL RTRIG_PON_C2 (CLK:=appoggio)      ** Appoggio

LD  Manual_alignment
AND appoggio
ST  Manual_align

CAL RTRIG_man_ali_C2(CLK:=Manual_align)

LD   RTRIG_PON_C2.Q
AND  (
LD   %ax34.ra4
SUB  %ax58.ra4
ABS
GT   200                 * threshold 1 dmm
AND (
 LD   %ax34.ra4
 SUB  %ax58.ra4
 ABS
 LE   %LSRCostK8
)
)
OR   RTRIG_man_ali_C2.Q
AND  MACC_TARATA                   ** (gPlc0.9)Assi tarati
AND  %ax34.ra3.0                    * Asse fermo teorico
AND  %ax58.ra3.0                    * Asse fermo teorico
ANDN PRGRUN_CN0                    ** M0.0 cn0.rc8.0  Programma in corso
S    start_alignment_C2

LD   start_alignment_C2
ST   POS_AX58.xax_ENABLE

LDN  POS_AX58.xax_ENABLE
OR   TP_PRGOFF_GEAR.Q
OR   TOF_RESET_GEAR.Q
ST   POS_AX58.xax_CLEAR

LD   POS_AX58.xax_ENABLE
AND  POS_AX58.yax_READY
ANDN POS_AX58.yax_ENDOK
ANDN POS_AX58.yax_ENDERR
ST   POS_AX58.xax_START

LD   %ax34.ra4
ST   POS_AX58.xax_QUOTA

LD   %pa9
ST   POS_AX58.xax_VEL

CAL  POS_AX58

LD   POS_AX58.yax_ENDOK
OR   POS_AX58.yax_ENDERR
OR   I_I_EMERGENZA                 ** Machine OK (no EMERG.)
***OR   EMER_GEN                      ** (M0.10)Emergenza generale
R    start_alignment_C2

LD   %ax34.ra4
SUB  %ax58.ra4
ABS
GT   %LSRCostK8
AND  PRGRUN_CN0                    ** M0.0 cn0.rc8.0  Programma in corso
ANDN %ServiceMillePGM.1
S   %PLCerr0.31                * Spindles not aligned

LD  Pul_Reset                      ** (gPlc0.3)Reset pushbutton
R   %PLCerr0.31                * Spindles not aligned

NOAX58:

LD  Pul_Reset                      ** (gPlc0.3)Reset pushbutton
R   GearingC_C1Off

***
* Gearing C-C2(GearingC_C1Off keeps same as C1)

LD   CMD_C_C2_UNLOCK
EQ   1
OR   GearingC_C1Off
ST   appoggio

CAL  TRIG_GEAR_C_C2(CLK:=appoggio)

LDN  EMER_GEN                      ** M0.10 Emergenza generale
AND  GESTAX58.xCloseLoop
ANDN POS_AX58.xax_ENABLE
ANDN ch5_in_ref                    ** channel 5 in ref
ST   appoggio

LD   appoggio
ANDN CMD_C_C2_UNLOCK
S    cmd_c_c2_gear_run

LD   spindle_geared_C2                ** axes gearing enable from function block
OR   CMD_C_C2_UNLOCK
R    cmd_c_c2_gear_run

CAL  TON_GEAR_C_C2(IN=appoggio,PT=800) ** Appoggio

LD   TON_GEAR_C_C2.Q
ANDN ch0_in_ref                    ** channel 0 in ref
ANDN BUP_JOGOPEN                   ** ui16.16 Selezione esecuzione JOG a loop aperto
AND (
LDN  CMD_C_C2_UNLOCK               ** M200 Unlock gearing C-C1
ANDN GearingC_C1Off
)
ST   GEAR_C_C2.xax_ENABLE          * ------> CONDIZ.RICHIESTA DI AGGANCIO

LDN  GEAR_C_C2.xax_ENABLE
OR   TRIG_GEAR_C_C2.Q
OR   TP_PRGOFF_GEAR.Q
OR   TOF_RESET_GEAR.Q
ST   GEAR_C_C2.xax_CLEAR

LD   GEAR_C_C2.xax_ENABLE
AND  GEAR_C_C2.yax_READY
ANDN GEAR_C_C2.yax_ENDOK
ANDN GEAR_C_C2.yax_ENDERR
ST   GEAR_C_C2.xax_START

LD   34
ST   GEAR_C_C2.xax_MASTER

LD   1                             * Modalit?di inseguimente(VA BENE LASCIARE SEMPRE 1)
ST   GEAR_C_C2.xax_TRNUM
ST   GEAR_C_C2.xax_TRDEN

CAL  GEAR_C_C2

LD   GEAR_C_C2.yax_RUNNING
AND  GEAR_C_C2.xax_ENABLE
S    spindle_geared_C2                ** axes gearing enable from function block

LDN  GEAR_C_C2.xax_ENABLE
OR   GEAR_C_C2.yax_ENDERR
R    spindle_geared_C2                ** axes gearing enable from function block

LDN  spindle_geared_C2                ** axes gearing enable from function block
ST   FBK_C_C2_UNLOCK               ** M201 Feedback gearing C-C1

**************************
* Acknowledg funzioni "M"
**************************
*
LD   %PLCFLAGS.0
ST   CH5END.xWaitMFun

CAL  CH5END

LD   M30010_CN3                    ** M0.6 Sblocco Richiesta servizio (M10000_CN0 inizialavorazione)
ORN  HEADZSEL                      ** (gPlc13.4)Testa 1 selezionata
OR(
LD   M30011_CN3                    ** M0.7 Sblocco Richiesta servizio (M10001_CN0 finelavorazione)
ORN  HEADZSEL                      ** (gPlc13.4)Testa 1 selezionata
)
ST   Appoggio                      ** Appoggio

CAL  R_TRIG30000(CLK=Appoggio)     ** FronteUp Sblocco Richiesta servizio per Unit_1

LD   M30010_CN3                    ** M0.6 Sblocco Richiesta servizio (M10000_CN0 inizialavorazione)
ORN  HEADZSEL                      ** (gPlc13.4)Testa 1 selezionata
S    UnlockCn0funzReq              ** Sblocco richiesta servizio da CN0 [(M10000 iniziolav.) / M10001(finelav.)]

LD   M30011_CN3                    ** M0.7 Sblocco Richiesta servizio (M10001_CN0 finelavorazione)
ORN  HEADZSEL                      ** (gPlc13.4)Testa 1 selezionata
ORN  PRGRUN_CN3                    ** M0.2 cn3.rc8.0  Programma in corso
R    UnlockCn0funzReq              ** Sblocco richiesta servizio da CN0 [(M10000 iniziolav.) / M10001(finelav.)]

*//============================================================================
*// CH6 CANALE COMPUTAZIONALE
*//============================================================================
CH6

*//============================================================================
*// CN7 Horizontal unloading supports channel
*//============================================================================
LD   GSTMAC.yChSelMask.7
AND  SEL_ASSE.yExtMask.2
ST   Sel_Z_Ch7

LD   GSTMAC.yChSelMask.7
AND  SEL_ASSE.yExtMask.3
ST   Sel_U_Ch7

LD   GSTMAC.yChSelMask.7
AND  SEL_ASSE.yExtMask.4
ST   Sel_V_Ch7

LD   GSTMAC.yChSelMask.7
AND  SEL_ASSE.yExtMask.5
ST   Sel_W_Ch7

CH7

*//============================================================================
*// CN8 Vertical unloading supports channel
*//============================================================================
LD   GSTMAC.yChSelMask.8
AND  SEL_ASSE.yExtMask.1
ST   Sel_Y_Ch8

LD   GSTMAC.yChSelMask.8
AND  SEL_ASSE.yExtMask.2
ST   Sel_Z_Ch8

LD   GSTMAC.yChSelMask.8
AND  SEL_ASSE.yExtMask.3
ST   Sel_U_Ch8

LD   GSTMAC.yChSelMask.8
AND  SEL_ASSE.yExtMask.4
ST   Sel_V_Ch8

LD   GSTMAC.yChSelMask.8
AND  SEL_ASSE.yExtMask.5
ST   Sel_W_Ch8

CH8

*//============================================================================
*// CN9 Loader Horizontal supports | Horizontal Following Clamps channel
*//============================================================================
LD   GSTMAC.yChSelMask.9
AND  SEL_ASSE.yExtMask.1
ST   Sel_Y_Ch9

LD   GSTMAC.yChSelMask.9
AND  SEL_ASSE.yExtMask.2
ST   Sel_Z_Ch9

LD   GSTMAC.yChSelMask.9
AND  SEL_ASSE.yExtMask.3
ST   Sel_U_Ch9

LD   GSTMAC.yChSelMask.9
AND  SEL_ASSE.yExtMask.4
ST   Sel_V_Ch9

CH9

*******************************************************************************
*   MACCEND MANAGEMENT
*******************************************************************************
LD   ALWAYS_ONE                    ** PLCFLAGS.1  Flag sempre stato on
ST   MACCEND.xEnabOvsAuto

CAL  MACCEND

LD   MACCEND.yAllDriveEn           * all drives are enable
ST   AllDriveEnable                ** All drives are enabled

LD   MACCEND.yAxStopped   * Assi fermi
ST   AxStopSincGRP                 ** (gPlc13.11)Assi Fermi per sincronismo GRP[ax]

LD   MACCEND.yZeroed
OR   (
LD   AxesAreAbsolute               ** (LsPlc47.19) All axes are absolute
AND  (
LD   GESTAX9.yZeroed
ORN  %cn0.cc1.5
)
)
ST   MACC_TARATA                   ** (gPlc0.9)Assi tarati

LD   MACCEND.yInAlarm               * Macchina in allarme
ST   MACC_ALARM                    ** (gPlc0.10)Macchina in allarme

*******************************************************************************
* Gestione RTCP tuning
*******************************************************************************
CAL TRIG_RTCPT(CLK=EnabJogTuning)  ** Jog tuning RTCP (UI)

LD   TRIG_RTCPT.Q        * Jog tuning RTCP (UI)
OR   EnJogRtcp                     ** (gPlc0.18)Abilitazione Jog RTCP tuning
AND(
LDN  TRIG_RTCPT.Q        * Jog tuning RTCP (UI)
ORN  EnJogRtcp                     ** (gPlc0.18)Abilitazione Jog RTCP tuning
)
AND  ch3_in_jog                    ** channel 3 in jog
ANDN ch3_in_aut                    ** channel 3 in aut
ST   EnJogRtcp                     ** (gPlc0.18)Abilitazione Jog RTCP tuning

***************************************
* Gestione registri  JOG RTCP/MX
* Inserito anche rc86 di cn4 perch?
* nel blocco funzione AxColl si
* riprogrammano i fine corsa SW degli assi
* Y 2 Y1 associati
* rispettivamente a cn0 e cn4.
***************************************

* Abilita M_JCR_SUBSYSTEM_ENABLE in JTX_CMDREG
LD   MACC_TARATA                   ** (gPlc0.9)Assi tarati
ST   %cn3.rc86.0
ST   %cn4.rc86.0

* M_JCR_MXM_USE_CURRENT in JTX_CMDREG
* Mettere a 1 se si vuole traslare con la matrice attiva (es.: rotaz pezzo)
LD   %PLCFLAGS.0
ST   %cn3.rc86.16
ST   %cn4.rc86.16

* Disabilita M_JCR_ENABLE_ABS_LS in JTX_CMDREG
LD   %PLCFLAGS.0
ST   %cn3.rc86.2
ST   %cn4.rc86.2

* Trasformazione selezionata da programma
LD   JOG_ENABLE                    ** (gPlc0.22)Jog Enable
ST   %cn3.rc86.20        * Trasformazione selezionata da programma

* Trasformazione utente
LD   EnJogRtcp                     ** (gPlc0.18)Abilitazione Jog RTCP tuning
ST   %cn3.rc86.11        * Abilita la selezione utente degli assi del canale
ST   %cn3.rc86.21        * Trasformazione utente

* Trasformazione cinematica utente
LD   1
ST   %cn3.rc87           * JTX_USER_RTCP_TWI

LD   1
ST   %cn3.rc88           * JTX_USER_RTCP_THD

LD   1
ST   %cn3.rc89           * JTX_USER_RTCP_CED

* Assi per matrice/assi cartesiani RTCP utente
LD   0
ST   %cn3.rc96           * JTX_USER_CHANNEL_X_SELECT

LD   1
ST   %cn3.rc97           * JTX_USER_CHANNEL_Y_SELECT

LD   2
ST   %cn3.rc98           * JTX_USER_CHANNEL_Z_SELECT

***************************************
* Interblocco comandi Jog con Matrici attive
* Assi fermi (Interblocco MatJog)
***************************************
LDN  JOGrunning                    ** One axis moving in JOG
AND  MACCEND.yAxStopped  * Assi Fermi
ORN  GESTCH3.xMatJog     * Ab. matrici dinamiche per il JOG (provv.)
ST   Appoggio                      ** Appoggio

CAL  TON_NOJOG(IN=Appoggio,PT=500) ** Assi fermi (Interblocco MatJog)

* Abilita Jog RTCP and JOG
LD   TON_NOJOG.Q         * Assi fermi (Interblocco MatJog)
ORN  EnJogRtcp                     ** (gPlc0.18)Abilitazione Jog RTCP tuning
ST   EnabJogRTCP                   ** Abilita Jog RTCP

*******************************************************************************

LD   Pon_XT1                       ** PON Axe X_T1
AND  Pon_YT1                       ** PON Axe Y_T1
AND  Pon_ax30                      ** PON Axe U (30)
AND  Pon_ax31                      ** PON Axe V (30)
AND  Pon_ax31                      ** PON Axe W (30)
AND  Pon_ZT1                       ** PON Axe Y_T1
AND  Pon_WLens                     ** PON Axe W_Lens
AND  Pon_C                         ** PON Axe C
AND  Pon_C1                        ** PON Axe C1
AND  Pon_A                         ** PON Axe A
AND  Pon_B                         ** PON Axe B
AND  Pon_Z_Follow                  ** PON Axe Z follower
**AND  Pon_PIPE                      ** PON Axe PIPE pipe axis
AND  Pon_UnSupp_71
AND  Pon_UnSupp_72
AND  Pon_UnSupp_73
AND  Pon_UnSupp_74
AND  Pon_UnSupp_75
AND  Pon_Z_Follow
AND  Pon_Z_Follow2
AND  Pon_Z_Follow3
AND  Pon_Z_Follow4
AND  Pon_UnSupp_81
AND  Pon_UnSupp_82
AND  Pon_UnSupp_83
AND  Pon_UnSupp_84
AND  Pon_UnSupp_85
AND  Pon_UnSupp_86
AND  Pon_UnSupp_87
AND  Pon_UnSupp_88
ST   Pon                           ** PON

* Uscita CNC OK
LD   GESTCH0.yChanReady  * Canale Ready
AND  GESTCH3.yChanReady  * Canale Ready
ST   O_O_CNC_OK                    ** CNC OK

***LD   LsrVrtcFcSoftware             ** (LsPlc0.31)Intervento Fc Sofware in lavorazione Laser
LD   %vrtc1.VrdwStatRegister1.2     * Upper mandatory position limit reached
OR   %vrtc1.VrdwStatRegister1.3     * Lower mandatory position limit reached
AND  %vrtc1.VrdwCtrlRegister0.1
S    %PLCerr0.10          * Fc Sofware Da VRTC in lavorazione

LD   Pul_Reset                     ** (gPlc0.3)Reset pushbutton
R    %PLCerr0.10          * Fc Sofware Da VRTC in lavorazione

* Canale 0 in blocco

LD   %cn0.rc63           * Stato canale
GE   14
AND(
LD   %cn0.rc63           * Stato canale
LE   17
)
AND(
LD   %cn0.rc18           * Codice errore canale
EQ   0
)
ANDN %cn0.rc8.3          * rc8.3  Canale in allarme
ANDN %cn0.rc0.1          * rc0.1  Emergenza
ST   Appoggio                      ** Appoggio

CAL  TON_ERRC0(IN=Appoggio, PT=10000) ** Canale 0 in blocco

LD   TON_ERRC0.Q         * Canale 0 in blocco
ST   %PLCerr0.11         * Canale 0 in blocco

* Emergenza generale

LD   EMER_GEN                      ** M0.10 Emergenza generale
ST   %PLCerr1.0          * Emergenza generale

LD   I_I_EMERGENZA
S    %PLCerr1.1          * Laser safe activated,reset to continue
LD   Pul_Reset
R    %PLCerr1.1          * Laser safe activated,reset to continue

***************************
* PON per singolo asse    *
***************************
LD   TON_ABIL.Q           * Abilitazione drives
ANDN Pon_ax30                      ** PON Axe U (30)
S    %PLCerr1.17

LD   TON_ABIL.Q           * Abilitazione drives
ANDN Pon_Mand             * PON Axe Mandrino
S    %PLCerr1.18          * Manca PON Axe Mandrino

LD   TON_ABIL.Q           * Abilitazione drives
ANDN Pon_XT1                       ** PON Axe X_T1
S    %PLCerr1.19          * Manca PON Axe X_T1

LD   TON_ABIL.Q           * Abilitazione drives
ANDN Pon_YT1                       ** PON Axe Y_T1
S    %PLCerr1.20          * Manca PON Axe Y_T1

LD   TON_ABIL.Q           * Abilitazione drives
ANDN Pon_ZT1                       ** PON Axe Y_T1
S    %PLCerr1.21          * Manca PON Axe Z_T1

LD   TON_ABIL.Q           * Abilitazione drives
ANDN Pon_WLens                     ** PON Axe W_Lens
S    %PLCerr1.28          * Power On Focal axis not present

LD   TON_ABIL.Q           * Abilitazione drives
ANDN Pon_C                         ** PON Axe C
S    %PLCerr1.29          * Power On C axis

LD   TON_ABIL.Q           * Abilitazione drives
ANDN Pon_C1                        ** PON Axe C1
S    %PLCerr1.30          * Power On C1 axis

*LD   TON_ABIL.Q           * Abilitazione drives
*ANDN Pon_PIPE             * PON Axe Pipe
*S    %PLCerr1.31          * Power On PIPE axis

LD   TON_ABIL.Q           * Abilitazione drives
ANDN Pon_Z_Follow            ** PON Axe X_T1
ST   %PLCerr2.13          * Power On Z follower axis

LD   TON_ABIL.Q           * Abilitazione drives
ANDN Pon_UnSupp_71
ST   %PLCerr3.0           * Power On Z follower axis

LD   TON_ABIL.Q           * Abilitazione drives
ANDN Pon_UnSupp_72
ST   %PLCerr3.1           * Power On Z follower axis

LD   TON_ABIL.Q           * Abilitazione drives
ANDN Pon_UnSupp_73
ST   %PLCerr3.2           * Power On Z follower axis

LD   TON_ABIL.Q           * Abilitazione drives
ANDN Pon_UnSupp_74
ST   %PLCerr3.3           * Power On Z follower axis

LD   TON_ABIL.Q           * Abilitazione drives
ANDN Pon_UnSupp_75
ST   %PLCerr3.4           * Power On Z follower axis

LD   TON_ABIL.Q           * Abilitazione drives
ANDN Pon_Z_Follow2
ST   %PLCerr3.10

LD   TON_ABIL.Q           * Abilitazione drives
ANDN Pon_Z_Follow
ST   %PLCerr3.12

LD   TON_ABIL.Q           * Abilitazione drives
ANDN Pon_Z_Follow3
ST   %PLCerr3.13

LD   TON_ABIL.Q           * Abilitazione drives
ANDN Pon_UnSupp_81
ST   %PLCerr3.14

LD   TON_ABIL.Q           * Abilitazione drives
ANDN Pon_UnSupp_82
ST   %PLCerr3.15

* Assi in allarme

LD   MACCEND.yInAlarm
OR   %PLCerr1.17          * Manca PON Axe Gantry
OR   %PLCerr1.18          * Manca PON Axe Mandrino
OR   %PLCerr1.19          * Manca PON Axe X_T1
OR   %PLCerr1.20          * Manca PON Axe Y_T1
OR   %PLCerr1.21          * Manca PON Axe Z_T1
OR   %PLCerr1.28          * Power On Focal axis not present
OR   %PLCerr1.29          * Power On C axis
OR   %PLCerr1.30          * Power On C1 axis
OR   %PLCerr1.31          * Power On PIPE axis
OR(
     LD   %PLCerr3
     NE   0
)
S    %PLCerr2.26          * Assi in allarme

LD   RESET_ALLARMI 		              ** M100.4  Cancellazione allarmi attiva
JMPCN STATE_CAN_ALLARM
LD   0
ST   %PLCerr1
ST   %PLCerr2
ST   %PLCerr3
STATE_CAN_ALLARM:

*==============================================================================
* W1-10 Copy Paste Management
*==============================================================================
* (1- 15) for page(4000-4014)
LD     %Uipl.Page
SUB    3999
ST     CurrentWPage

LD     Btn_Cpy_W
ANDN   %cn0.rc8.0
ANDN   Aux_Req_CpyW
AND(
LD     CurrentWPage
GE     1
)
AND(
LD     CurrentWPage
LE     15
)
ST     appoggio
CAL    TP_CpyW(IN:=appoggio,PT:=1000)
LD     TP_CpyW.Q
ST     Aux_Req_CpyW

************************************************************
*                 Condizioni di emergenza                  *
************************************************************
LD   %PLCerr0
NE   0
OR (
LD   %PLCerr2
NE   0
)
OR   %PLCerr1.4                    * Manca aria compressa
OR   %PLCerr20.22
OR   %PLCerr20.23
OR   %PLCerr20.24
OR   %PLCerr20.25
OR   %PLCerr20.26
ORN  MACCHINA_OK                   ** M100.1  Macchina OK
ANDN Pul_Reset                     ** (gPlc0.3)Reset pushbutton
ST   EMER_GEN                      ** M0.10 Emergenza generale

LD   Pul_Reset                     ** (gPlc0.3)Reset pushbutton
JMPCN CANCELLA
LD   0
ST   %PLCerr0
ST   %PLCerr2
CANCELLA:

*******************************************************************************
*   Messaggi WARNING
*******************************************************************************

LD   TOF_RESET.Q         * Reset
ST   %PLCmsg0.0          * Reset in corso

***

LD   GESTAX0.xHoldMoving * Richiesta blocco avanzamento
OR   GESTAX1.xHoldMoving * Richiesta blocco avanzamento
OR   GESTAX6.xHoldMoving * Richiesta blocco avanzamento
OR   GESTAX27.xHoldMoving * Richiesta blocco avanzamento
OR   GESTAX28.xHoldMoving * Richiesta blocco avanzamento
OR   GESTAX30.xHoldMoving * Richiesta blocco avanzamento
ST   %PLCmsg0.1          ** block active feed X-Y

***

LD   PhotocellsOn                  ** (gPlc2.15)Photocells on
ST   %PLCmsg0.7          * Photocells msg

***

* Manuale in corso
LD   JOGrunning                    ** One axis moving in JOG
ST   %PLCmsg0.21         * Manuale in corso

* Taratura in corso
LD   REFrunning                    ** One axis moving in REF
ST   %PLCmsg0.22         * Taratura in corso
ST   REF_RUN                       ** M0.12 Taratura in corso

* Pos. incrementale in corso
LD   INCrunning                    ** One axis moving in INC
ST   %PLCmsg0.23         * Pos. incrementale in corso

* Assi non tarati
LDN  MACC_TARATA                   ** (gPlc0.9)Assi tarati
ST   %PLCmsg0.26         * Assi non tarati

* Ciclo automatico sospeso
LD   PRGSTOP_CN0                   ** (cn0.rc8.1)  Programma interrotto CN0
ST   %PLCmsg1.0          * Ciclo automatico sospeso

* Attesa start
LD   GESTCH0.yWaitMFun
ST   %PLCmsg1.16         * Attesa start

LDN  spindle_geared                ** axes gearing enable from function block
ST   %PLCmsg1.15

********************************************************************************
* Pipe and Plane Machine

*******************************************************************************
* PLC user function to commands and output overwriting
*******************************************************************************
LASER_OUT

*******************************************************************************
*END  USER MANAGEMENT
*******************************************************************************
*Gestione Output e segnali ESA->USR
#ifndef SIM_IO
OUT_CONFIG
#endif

*Gestione logica finale USR
USR_END

*********************************************************************************
* XXX Risolve il problema RESET dopo RETRACE IND
*********************************************************************************
LDN  %cn0.rc64.25       ** rc64.25 Comando forward retrace
ANDN %cn0.rc64.26       ** rc64.26 Comando reverse retrace
ST   %cn0.rc64.27       ** svuota code comandi
*******************************************************************************

LDN  PRGRUN_CN0                                  ** M10.8 Program running on Channel 0
JMPCN END
LD -1
ST Unlock_Channels
END:

USERLOGGER

NO_EXECUTE_PLC:
END_FUNCTION
